// TwinCAT 3 PLC project Untitled1
// ProgramVersion: 3.1.4026.12
// libraries:
//   Tc2_Standard, * (Beckhoff Automation GmbH)
//   Tc2_System, * (Beckhoff Automation GmbH)
//   Tc3_Module, * (Beckhoff Automation GmbH)
// project tree:
//   / PlcTask.TcTTO
//   POUs/ FB_OpenDichtKlep.TcPOU, MAIN.TcPOU
// real-time tasks:
//   TASK PlcTask: cycle T#10ms, priority 20, ADS port 350

CONFIGURATION Untitled1
    RESOURCE PLC ON TwinCAT3
        TASK PlcTask(INTERVAL := T#10ms, PRIORITY := 20);
        PROGRAM MAIN WITH PlcTask : MAIN;
    END_RESOURCE
END_CONFIGURATION

// ---- POUs/MAIN.TcPOU
PROGRAM MAIN
VAR
	fbCoalDrill 	: FB_Drill ; 
	fbcopperDrill	: FB_Drill ;
	fbIronDrill		: FB_Drill ;
	test : int;
		
	iCoalStash 		: UINT ; // total amount of coal
	iCopperOreStash : UINT ; // total amount of copper stored
	iIronOreStash	: UINT ; // Total amount of iron ore stash  
	
	fbIronProduction_1 		: FB_StoneFurnace;
	fbCopperProduction_1	: FB_StoneFurnace;
	
END_VAR


CollectOre();
ProduceIron();
CollectCopperOre();
test:=1;

METHOD CollectCopperOre : BOOL
VAR_INPUT
END_VAR
	fbCopperProduction_1();
END_METHOD

METHOD CollectOre : BOOL
VAR_INPUT
END_VAR
// run Drills
	fbCoalDrill(); 
	fbcopperDrill();
	fbIronDrill();

// collect ore
	iCoalStash 		:= iCoalStash + fbCoalDrill.ProductsOut;
	iCopperOreStash := iCopperOreStash + fbcopperDrill.ProductsOut;
	iIronOreStash	:= iIronOreStash + fbIronDrill.ProductsOut;
END_METHOD

METHOD ProduceIron : BOOL
VAR_INPUT
END_VAR

// run production
	fbIronProduction_1();
END_METHOD

END_PROGRAM

// ---- POUs/FB_OpenDichtKlep.TcPOU
FUNCTION_BLOCK FB_OpenDichtKlep IMPLEMENTS ITF_OpenDichtKlep
VAR
    tagName : STRING;
    inputOpen : ITF_DigIn;
	inputClosed : ITF_DigIn;
	output : ITF_DigOut;
	
	feedbackOpen : BOOL := FALSE;
	feedbackClosed : BOOL := FALSE;
	feedbackError : BOOL := FALSE;
	
	manOpen : BOOL := FALSE;
	manClose : BOOL := FALSE;

	currentMode : E_Bedrijfstoestand := E_Bedrijfstoestand.off;
	currentState : E_OpenDichtKlepState := E_OpenDichtKlepState.closed;
	expectedState : E_OpenDichtKlepState := E_OpenDichtKlepState.closed;
	
	timeOut : TON;
	errorTrigger : R_TRIG;
END_VAR

IF currentMode = E_Bedrijfstoestand.off THEN
	output.set(FALSE);
	expectedState := E_OpenDichtKlepState.closed;
END_IF

IF currentMode = E_Bedrijfstoestand.manual THEN
	IF manOpen THEN
		openManual();
		manOpen:= FALSE;
	END_IF
	IF manClose THEN
		closeManual();
		manClose:= FALSE;
	END_IF
END_IF

feedbackOpen := inputOpen.get() AND NOT inputClosed.get();
feedbackClosed := inputClosed.get() AND NOT inputOpen.get();
feedbackError := inputClosed.get() AND inputOpen.get();

timeOut(IN := NOT(expectedState = currentState), PT := T#5S);
errorTrigger(CLK := (timeOut.Q OR feedbackError));

IF errorTrigger.Q THEN
	currentState := E_OpenDichtKlepState.error;
	main.alarms.append(tag := tagName, msg := 'Klepstoring gedetecteerd');
END_IF

CASE expectedState OF
E_OpenDichtKlepState.closed :
	IF feedbackClosed THEN
		currentState := E_OpenDichtKlepState.closed;
	ELSIF NOT(currentState = E_OpenDichtKlepState.error) THEN
		currentState := E_OpenDichtKlepState.closing;
	END_IF
E_OpenDichtKlepState.open :
	IF feedbackOpen THEN
		currentState := E_OpenDichtKlepState.open;
	ELSIF NOT(currentState = E_OpenDichtKlepState.error) THEN
		currentState := E_OpenDichtKlepState.opening;
	END_IF
END_CASE

METHOD close : BOOL
VAR_INPUT
END_VAR
IF currentMode = E_Bedrijfstoestand.auto THEN
	output.set(FALSE);
	expectedState := E_OpenDichtKlepState.closed;
	close := TRUE;
ELSE
	close := FALSE;
END_IF
END_METHOD

METHOD closeManual : BOOL
VAR_INPUT
END_VAR
IF currentMode = E_Bedrijfstoestand.manual THEN
	output.set(FALSE);
	expectedState := E_OpenDichtKlepState.closed;
	closeManual := TRUE;
ELSE
	closeManual := FALSE;
END_IF
END_METHOD

METHOD FB_init : BOOL
VAR_INPUT
	bInitRetains : BOOL; // if TRUE, the retain variables are initialized (warm start / cold start)
	bInCopyCode : BOOL;  // if TRUE, the instance afterwards gets moved into the copy code (online change)
	tag : STRING;
	DigInClosed : ITF_DigIn;
	DigInOpened : ITF_DigIn;
	DigOut : ITF_DigOut;
END_VAR
tagname := tag;
inputClosed := DigInClosed;
inputOpen := DigInOpened;
output := DigOut;
END_METHOD

METHOD open : BOOL
VAR_INPUT
END_VAR
IF currentMode = E_Bedrijfstoestand.auto THEN
	output.set(TRUE);
	expectedState := E_OpenDichtKlepState.open;
	open := TRUE;
ELSE
	open := FALSE;
END_IF
END_METHOD

METHOD openManual : BOOL
VAR_INPUT
END_VAR
IF currentMode = E_Bedrijfstoestand.manual THEN
	output.set(TRUE);
	expectedState := E_OpenDichtKlepState.open;
	openManual := TRUE;
ELSE
	openManual := FALSE;
END_IF
END_METHOD

PROPERTY state : E_OpenDichtKlepState
GET
state := currentState;
END_GET
END_PROPERTY

END_FUNCTION_BLOCK
